PROGRAM Reservoir
VAR
	fbLevelCtrl : LevelControl;
	bLowLevelAlarm : BOOL;
	bHighLevelAlarm : BOOL;
	
	bResetButton : BOOL;
	bStartButton : BOOL;
	bStopButton : BOOL;
	
	bPumpLight : BOOL;
	bAgitatorLight : BOOL;
	bSolenoidALight : BOOL;
	bSolenoidBLight : BOOL;
	
	rSensorInput : REAL;
	
	rPumpOutput : LREAL;
	rAgitatorOutput : LREAL;
END_VAR

bLowLevelAlarm := fbLevelCtrl.bLowLevel;
bHighLevelAlarm := fbLevelCtrl.bHighLevel;

fbLevelCtrl.bStart := bStartButton;
fbLevelCtrl.bStop := bStopButton;
fbLevelCtrl.bReset := bResetButton;

bPumpLight := fbLevelCtrl.bPump;
bAgitatorLight := fbLevelCtrl.bAgitator;
bSolenoidALight := fbLevelCtrl.bSolenoidA;
bSolenoidBLight := fbLevelCtrl.bSolenoidB;

fbLevelCtrl.rWaterLevel := rSensorInput;

rPumpOutput := fbLevelCtrl.rPumpPos;
rAgitatorOutput := fbLevelCtrl.rAgitatorPos;


fbLevelCtrl();

END_PROGRAM

(* stored: Version 1.1.0.1, ProductVersion 3.1.4024.12
   POU Reservoir: Id {3baf05ff-c014-4d1e-aa96-04828a5fe1b5}, SpecialFunc None *)
